// TIA Portal V20 export
TYPE "typeStationDataUnwidnerInfeed"
   STRUCT
      "Unwind Tension Set Point 1" : Real;   // MPa
      "Unwind Tension Actual 1" : Real;   // N
      "Unwind Roll Diameter 1" : Real;   // mm
      "Unwind Roll Diameter 2" : Real;   // mm
      "Bobbin ID 1" : String;   // N/A
      "Bobbin ID 2" : String;   // N/A
      "Cycle end Trigger" : Bool;   // I/O
      Blocked : Bool;   // I/O
      Starved : Bool;   // I/O
      "Good Count" : DInt;   // Cnt
      "Reject Count" : DInt;   // Cnt
      "Fault bit" : Bool;   // I/O
      Fault : Bool;   // I/O
      PUN : String;   // N/A
      "Part Type" : String;   // N/A
      "FTQ & Reject code" : String;   // N/A
   END_STRUCT;
END_TYPE
